// TIA Portal V16 export
// export: Created 2022-02-04T14:40:20.5072516Z, ExportSetting WithDefaults, DisplayName Totally Integrated Automation Portal, DisplayVersion V16 Update 1, DisplayName TIA Portal Version Control Interface, DisplayVersion V16, DisplayName TIA Portal Openness, DisplayVersion V16, DisplayName SINAMICS Startdrive Advanced, DisplayVersion V16 Update 5, DisplayName SINAMICS Startdrive G130, G150, S120, S150, SINAMICS MV, S210, DisplayVersion V16 Update 5, DisplayName SINAMICS Startdrive G110M, G120, G120C, G120D, G120P, G115D, DisplayVersion V16 Update 5, DisplayName STEP 7 Professional, DisplayVersion V16, DisplayName STEP 7 Safety, DisplayVersion V16, DisplayName WinCC Advanced, DisplayVersion V16, DisplayName SIMATIC Visualization Architect, DisplayVersion V16
DATA_BLOCK "EvaluationZoneThrowOFF_DB"   // DB22
VERSION : 0.1
// stored: AutoNumber true, InstanceOfName EvaluationZoneThrowOFF, InstanceOfType FB
"EvaluationZoneThrowOFF"
   // VAR_INPUT
   //    StartEvaluationArea : Bool;
   //    EndEvaluationArea : Bool;
   //    DefectSignal : Bool;
   //    MU_mode : Bool;
   //    DropArea : Bool;
   //    Reset : Bool;
   // END_VAR
   // VAR_OUTPUT
   //    DefectDrop_CMD_UP : Bool;
   //    DefectDrop_CMD_DOWN : Bool;
   //    CommonAlarmEvaluationZone : Bool;
   //    AlarmBoardNotExitFromZone : Bool;
   //    FaultQueueOverflow : Bool;
   //    FaultGhostBoard : Bool;
   // END_VAR
   // VAR RETAIN
   //    StartEvaluationArea_old : Bool;
   //    EndEvaluationArea_old : Bool;
   //    DropArea_old : Bool;
   //    CanEvaluate : Bool;
   //    CMD_up_old : Bool;
   //    BoardIterator : Int;
   //    SolutionQueue : Array[0..7] of Bool;
   // END_VAR
BEGIN
END_DATA_BLOCK
